TYPE (* Color for all states *)
  (* Description: Copyright (c) 2025 HR Agrartechnik GmbH This program and the accompanying materials are made available under the terms of the Eclipse Public License 2.0 which is available at https://www.eclipse.org/legal/epl-2.0/ SPDX-License-Identifier: EPL-2.0 *)
  (* Version 1.0, 2025-06-11, Franz Höpfinger, HR Agrartechnik GmbH *)
  PACKAGE logiBUS::utils::sequence::schieber;
  IMPORT isobus::UT::Q::const::colours::COLOR_WHITE;
  SchieberColorStruct : STRUCT
    Unknown : USINT := COLOR_WHITE; (* u8Colour for Unknown State *)
    Closed : USINT := COLOR_WHITE; (* u8Colour for Closed State *)
    Opening : USINT := COLOR_WHITE; (* u8Colour for Opening State *)
    Opened : USINT := COLOR_WHITE; (* u8Colour for Opened State *)
    Closing : USINT := COLOR_WHITE; (* u8Colour for Closing State *)
  END_STRUCT;
END_TYPE
